Fanuc KAREL source: kt00936.KL

-- PROVISIONAL review KL for V1013-1; original PC SHA256 c46bf99fb7b598f0708cb578b2da145081b6a94d4005f7462c45c676849c1f29
-- Incomplete behavior may be omitted. Consult companion uncertainty JSON. Do not deploy.
PROGRAM KT00936
%NOLOCKGROUP
VAR
  ENTRY : INTEGER
  PNAME : STRING[80]
  VNAME : STRING[80]
  STATUS : INTEGER
  VALUE : STRING[80]
BEGIN
  -- UNRESOLVED_PC offsets 5-12; opcodes 9C,23
  -- UNRESOLVED_PC offsets 17-25; opcodes 3F,75
  -- UNRESOLVED_PC offsets 30-43; opcodes 3F,75
  -- UNRESOLVED_PC offsets 48-88; opcodes 27,22,22,2A,22,2A,22,2A,22,AF
  -- UNRESOLVED_PC offsets 93-97; opcodes 7F
END KT00936
